ABB RobotStudio station: ProiectSCR.rspag

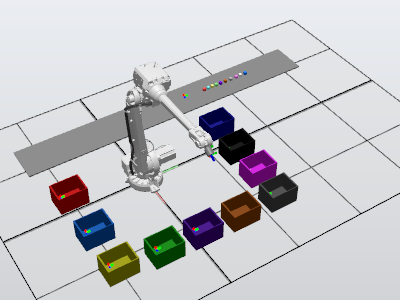
--- station ---
Station Tema1_SCR_Grigore_Vlad (saved by RobotStudio 24.3.10958.1)
Controller IRB4600_20_250
  mechanical unit ROB_1: IRB4600_20_250_C_01, 6 joints, base frame (0, 0, 0) mm
Layout (positions relative to the parent item):
  - IRB4600_20_250_C_01 [mechanism, from %ABB.RobotStudio.Models.IRB4600%\IRB4600_20_250_C_G_01.rslib] at (0, 0, 0) mm; joint values [0, 0, 0, 0, 0.5236, 0] (rad or m)
  - Container_1 [part] at (-320.44, -1190.22, 30) mm, size 300 x 400 x 270 mm
  - Banda [part] at (-1428.04, -1283.76, 0) mm, size 550 x 4550 x 20 mm
  - Pachet_1 [part] at (-1164.97, 1677.25, 60) mm, rotated rx 180 ry 0 rz 180 deg, size 40 x 40 x 40 mm
  - Container_2 [part] at (386.4, -1190.22, 30) mm, size 300 x 400 x 270 mm
  - Container_3 [part] at (1012.12, -1190.22, 30) mm, size 300 x 400 x 270 mm
  - Container_4 [part] at (1087.87, -610.7, 30) mm, size 300 x 400 x 270 mm
  - Container_6 [part] at (1101.15, 485.48, 30) mm, size 300 x 400 x 270 mm
  - Container_7 [part] at (1088.83, 1073.15, 30) mm, size 300 x 400 x 270 mm
  - Container_8 [part] at (596.46, 1111.34, 30) mm, size 300 x 400 x 270 mm
  - Container_9 [part] at (89.93, 1120.66, 30) mm, size 300 x 400 x 270 mm
  - Container_10 [part] at (-439.15, 1146.37, 30) mm, size 300 x 400 x 270 mm
  - MyNewTool [mechanism] at (1479.11, 0, 1722.5) mm, rotated rx 180 ry 60 rz 180 deg
      TCP MyNewTool at (0, 0, 80) mm
      links: Part_2
  - Container_5 [part] at (1087.87, -64.6, 30) mm, size 300 x 400 x 270 mm
  - Pachet_3 [part] at (-1164.97, 1820.33, 60) mm, rotated rx 180 ry 0 rz 180 deg, size 40 x 40 x 40 mm
  - Pachet_5 [part] at (-1164.97, 1973.31, 60) mm, rotated rx 180 ry 0 rz 180 deg, size 40 x 40 x 40 mm
  - Pachet_6 [part] at (-1164.97, 2058.75, 60) mm, rotated rx 180 ry 0 rz 180 deg, size 40 x 40 x 40 mm
  - Pachet_7 [part] at (-1164.97, 2158.23, 60) mm, rotated rx 180 ry 0 rz 180 deg, size 40 x 40 x 40 mm
  - Pachet_8 [part] at (-1164.97, 2259.91, 60) mm, rotated rx 180 ry 0 rz 180 deg, size 40 x 40 x 40 mm
  - Pachet_10 [part] at (-1164.97, 2429.71, 60) mm, rotated rx 180 ry 0 rz 180 deg, size 40 x 40 x 40 mm
  - Pachet_4 [part] at (-1164.97, 1892.62, 60) mm, rotated rx 180 ry 0 rz 180 deg, size 40 x 40 x 40 mm
  - Pachet_9 [part] at (-1164.97, 2336.17, 60) mm, rotated rx 180 ry 0 rz 180 deg, size 40 x 40 x 40 mm
  - SmartComponent_1 [smart component]
      signals: DI Get, DI DeleteAll
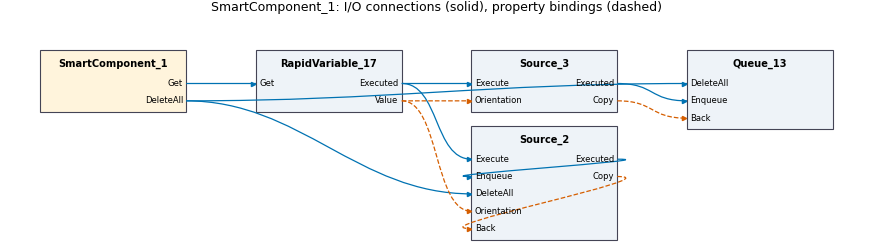
      connections:
        SmartComponent_1.Get -> RapidVariable_17.Get
        RapidVariable_17.Executed -> Source_2.Execute
        Source_2.Executed -> Queue_12.Enqueue
        SmartComponent_1.DeleteAll -> Queue_12.DeleteAll
        SmartComponent_1.DeleteAll -> Queue_13.DeleteAll
        Source_3.Executed -> Queue_13.Enqueue
        RapidVariable_17.Executed -> Source_3.Execute
        RapidVariable_17.Value => Source_2.Orientation
        Source_2.Copy => Queue_12.Back
        RapidVariable_17.Value => Source_3.Orientation
        Source_3.Copy => Queue_13.Back
    - RapidVariable_17 [smart component, from Components\RapidVariable.rslib]
        properties: DataType=orient; Controller=IRB4600_20_250; Task=T_ROB1; Module=Module1; Variable=RotXYZ; Value=[3.14159265358979 1.08734199990513E-38 3.14159265358979]
    - Source_3 [smart component, from Components\Source.rslib]
        properties: Source=Pachet_1; Copy=(none); Parent=(none); Position=[-1.164969 1.332694 0.06]; Orientation=[3.14159265358979 1.08734199990513E-38 3.14159265358979]; Transient=false; PhysicsBehavior=-1
    - Queue_13 [smart component, from Components\Queue.rslib]
        properties: Back=(none); Front=(none); Queue=; NumberOfObjects=0
  - SmartComponent_2 [smart component]
      signals: DI Get, DI DeleteAll
      connections:
        SmartComponent_2.Get -> RapidVariable_17.Get
        RapidVariable_17.Executed -> Source_2.Execute
        Source_2.Executed -> Queue_12.Enqueue
        SmartComponent_2.DeleteAll -> Queue_12.DeleteAll
        RapidVariable_17.Executed -> Source_4.Execute
        Source_4.Executed -> Queue_12.Enqueue
        RapidVariable_17.Value => Source_2.Orientation
        Source_2.Copy => Queue_12.Back
        RapidVariable_17.Value => Source_4.Orientation
        Source_4.Copy => Queue_12.Back
    - RapidVariable_17 [smart component, from Components\RapidVariable.rslib]
        properties: DataType=orient; Controller=IRB4600_20_250; Task=T_ROB1; Module=Module1; Variable=RotXYZ; Value=[3.14159265358979 1.08734199990513E-38 3.14159265358979]
    - Queue_12 [smart component, from Components\Queue.rslib]
        properties: Back=(none); Front=(none); Queue=; NumberOfObjects=0
    - Source_4 [smart component, from Components\Source.rslib]
        properties: Source=Pachet_2; Copy=(none); Parent=(none); Position=[-1.164969 1.332694 0.06]; Orientation=[3.14159265358979 1.08734199990513E-38 3.14159265358979]; Transient=false; PhysicsBehavior=-1
  - SmartComponent_3 [smart component]
      signals: DI Get, DI DeleteAll
      connections:
        SmartComponent_3.Get -> RapidVariable_17.Get
        RapidVariable_17.Executed -> Source_2.Execute
        Source_2.Executed -> Queue_12.Enqueue
        SmartComponent_3.DeleteAll -> Queue_12.DeleteAll
        RapidVariable_17.Value => Source_2.Orientation
        Source_2.Copy => Queue_12.Back
    - Source_2 [smart component, from Components\Source.rslib]
        properties: Source=Pachet_3; Copy=(none); Parent=(none); Position=[-1.164969 1.332694 0.06]; Orientation=[3.14159265358979 1.08734199990513E-38 3.14159265358979]; Transient=false; PhysicsBehavior=-1
    - RapidVariable_17 [smart component, from Components\RapidVariable.rslib]
        properties: DataType=orient; Controller=IRB4600_20_250; Task=T_ROB1; Module=Module1; Variable=RotXYZ; Value=[3.14159265358979 1.08734199990513E-38 3.14159265358979]
    - Queue_12 [smart component, from Components\Queue.rslib]
        properties: Back=(none); Front=(none); Queue=; NumberOfObjects=0
  - SmartComponent_4 [smart component]
      signals: DI Get, DI DeleteAll
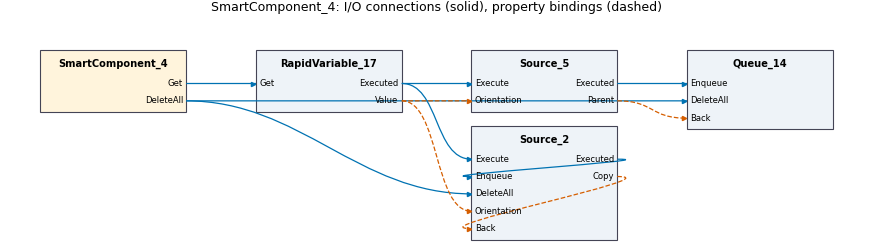
      connections:
        SmartComponent_4.Get -> RapidVariable_17.Get
        RapidVariable_17.Executed -> Source_2.Execute
        Source_2.Executed -> Queue_12.Enqueue
        SmartComponent_4.DeleteAll -> Queue_12.DeleteAll
        RapidVariable_17.Executed -> Source_5.Execute
        Source_5.Executed -> Queue_14.Enqueue
        SmartComponent_4.DeleteAll -> Queue_14.DeleteAll
        RapidVariable_17.Value => Source_2.Orientation
        Source_2.Copy => Queue_12.Back
        RapidVariable_17.Value => Source_5.Orientation
        Source_5.Parent => Queue_14.Back
    - RapidVariable_17 [smart component, from Components\RapidVariable.rslib]
        properties: DataType=orient; Controller=IRB4600_20_250; Task=T_ROB1; Module=Module1; Variable=RotXYZ; Value=[0 0 0]
    - Source_5 [smart component, from Components\Source.rslib]
        properties: Source=Pachet_4; Copy=(none); Parent=(none); Position=[-1.164969 1.332694 0.06]; Orientation=[0 0 0]; Transient=false; PhysicsBehavior=-1
    - Queue_14 [smart component, from Components\Queue.rslib]
        properties: Back=(none); Front=(none); Queue=; NumberOfObjects=0
  - SmartComponent_5 [smart component]
      signals: DI Get, DI DeleteAll
      connections:
        SmartComponent_5.Get -> RapidVariable_17.Get
        RapidVariable_17.Executed -> Source_2.Execute
        Source_2.Executed -> Queue_12.Enqueue
        SmartComponent_5.DeleteAll -> Queue_12.DeleteAll
        RapidVariable_17.Executed -> Source_6.Execute
        Source_6.Executed -> Queue_15.Enqueue
        SmartComponent_5.DeleteAll -> Queue_15.DeleteAll
        RapidVariable_17.Value => Source_2.Orientation
        Source_2.Copy => Queue_12.Back
        Source_6.Copy => Queue_15.Back
        RapidVariable_17.Value => Source_6.Orientation
    - RapidVariable_17 [smart component, from Components\RapidVariable.rslib]
        properties: DataType=orient; Controller=IRB4600_20_250; Task=T_ROB1; Module=Module1; Variable=RotXYZ; Value=[0 0 0]
    - Source_6 [smart component, from Components\Source.rslib]
        properties: Source=Pachet_5; Copy=(none); Parent=(none); Position=[-1.164969 1.332694 0.06]; Orientation=[0 0 0]; Transient=false; PhysicsBehavior=-1
    - Queue_15 [smart component, from Components\Queue.rslib]
        properties: Back=(none); Front=(none); Queue=; NumberOfObjects=0
  - SmartComponent_6 [smart component]
      signals: DI Get, DI DeleteAll
      connections:
        SmartComponent_6.Get -> RapidVariable_17.Get
        RapidVariable_17.Executed -> Source_2.Execute
        Source_2.Executed -> Queue_12.Enqueue
        SmartComponent_6.DeleteAll -> Queue_12.DeleteAll
        RapidVariable_17.Executed -> Source_7.Execute
        Source_7.Executed -> Queue_16.Enqueue
        SmartComponent_6.DeleteAll -> Queue_16.DeleteAll
        RapidVariable_17.Value => Source_2.Orientation
        Source_2.Copy => Queue_12.Back
        Source_7.Copy => Queue_16.Back
        RapidVariable_17.Value => Source_7.Orientation
    - RapidVariable_17 [smart component, from Components\RapidVariable.rslib]
        properties: DataType=orient; Controller=IRB4600_20_250; Task=T_ROB1; Module=Module1; Variable=RotXYZ; Value=[0 0 0]
    - Source_7 [smart component, from Components\Source.rslib]
        properties: Source=Pachet_6; Copy=(none); Parent=(none); Position=[-1.164969 1.332694 0.06]; Orientation=[0 0 0]; Transient=false; PhysicsBehavior=-1
    - Queue_16 [smart component, from Components\Queue.rslib]
        properties: Back=(none); Front=(none); Queue=; NumberOfObjects=0
  - SmartComponent_7 [smart component]
      signals: DI Get, DI DeleteAll
      connections:
        SmartComponent_7.Get -> RapidVariable_17.Get
        RapidVariable_17.Executed -> Source_2.Execute
        Source_2.Executed -> Queue_12.Enqueue
        SmartComponent_7.DeleteAll -> Queue_12.DeleteAll
        RapidVariable_17.Executed -> Source_8.Execute
        Source_8.Executed -> Queue_17.Enqueue
        SmartComponent_7.DeleteAll -> Queue_17.DeleteAll
        RapidVariable_17.Value => Source_2.Orientation
        Source_2.Copy => Queue_12.Back
        Source_8.Copy => Queue_17.Back
        RapidVariable_17.Value => Source_8.Orientation
    - RapidVariable_17 [smart component, from Components\RapidVariable.rslib]
        properties: DataType=orient; Controller=IRB4600_20_250; Task=T_ROB1; Module=Module1; Variable=RotXYZ; Value=[0 0 0]
    - Source_8 [smart component, from Components\Source.rslib]
        properties: Source=Pachet_7; Copy=(none); Parent=(none); Position=[-1.164969 1.332694 0.06]; Orientation=[0 0 0]; Transient=false; PhysicsBehavior=-1
    - Queue_17 [smart component, from Components\Queue.rslib]
        properties: Back=(none); Front=(none); Queue=; NumberOfObjects=0
  - SmartComponent_8 [smart component]
      signals: DI Get, DI DeleteAll
      connections:
        SmartComponent_8.Get -> RapidVariable_17.Get
        RapidVariable_17.Executed -> Source_2.Execute
        Source_2.Executed -> Queue_12.Enqueue
        SmartComponent_8.DeleteAll -> Queue_12.DeleteAll
        RapidVariable_17.Executed -> Source_10.Execute
        Source_10.Executed -> Queue_18.Enqueue
        SmartComponent_8.DeleteAll -> Queue_18.DeleteAll
        RapidVariable_17.Value => Source_2.Orientation
        Source_2.Copy => Queue_12.Back
        RapidVariable_17.Value => Source_10.Orientation
        Source_10.Copy => Queue_18.Back
    - RapidVariable_17 [smart component, from Components\RapidVariable.rslib]
        properties: DataType=orient; Controller=IRB4600_20_250; Task=T_ROB1; Module=Module1; Variable=RotXYZ; Value=[0 0 0]
    - Source_10 [smart component, from Components\Source.rslib]
        properties: Source=Pachet_8; Copy=(none); Parent=(none); Position=[-1.164969 1.332694 0.06]; Orientation=[0 0 0]; Transient=false; PhysicsBehavior=-1
    - Queue_18 [smart component, from Components\Queue.rslib]
        properties: Back=(none); Front=(none); Queue=; NumberOfObjects=0
  - SmartComponent_9 [smart component]
      signals: DI Get, DI DeleteAll
      connections:
        SmartComponent_9.Get -> RapidVariable_17.Get
        RapidVariable_17.Executed -> Source_2.Execute
        Source_2.Executed -> Queue_12.Enqueue
        SmartComponent_9.DeleteAll -> Queue_12.DeleteAll
        RapidVariable_17.Executed -> Source_11.Execute
        Source_11.Executed -> Queue_19.Enqueue
        SmartComponent_9.DeleteAll -> Queue_19.DeleteAll
        RapidVariable_17.Value => Source_2.Orientation
        Source_2.Copy => Queue_12.Back
        Source_11.Copy => Queue_19.Back
        RapidVariable_17.Value => Source_11.Orientation
    - RapidVariable_17 [smart component, from Components\RapidVariable.rslib]
        properties: DataType=orient; Controller=IRB4600_20_250; Task=T_ROB1; Module=Module1; Variable=RotXYZ; Value=[0 0 0]
    - Source_11 [smart component, from Components\Source.rslib]
        properties: Source=Pachet_9; Copy=(none); Parent=(none); Position=[-1.164969 1.332694 0.06]; Orientation=[0 0 0]; Transient=false; PhysicsBehavior=-1
    - Queue_19 [smart component, from Components\Queue.rslib]
        properties: Back=(none); Front=(none); Queue=; NumberOfObjects=0
  - SmartComponent_10 [smart component]
      signals: DI Get, DI DeleteAll
      connections:
        SmartComponent_10.Get -> RapidVariable_17.Get
        RapidVariable_17.Executed -> Source_2.Execute
        Source_2.Executed -> Queue_12.Enqueue
        SmartComponent_10.DeleteAll -> Queue_12.DeleteAll
        RapidVariable_17.Executed -> Source_13.Execute
        Source_13.Executed -> Queue_20.Enqueue
        SmartComponent_10.DeleteAll -> Queue_20.DeleteAll
        RapidVariable_17.Value => Source_2.Orientation
        Source_2.Copy => Queue_12.Back
        Source_13.Copy => Queue_20.Back
        RapidVariable_17.Value => Source_13.Orientation
    - RapidVariable_17 [smart component, from Components\RapidVariable.rslib]
        properties: DataType=orient; Controller=IRB4600_20_250; Task=T_ROB1; Module=Module1; Variable=RotXYZ; Value=[0 0 0]
    - Source_13 [smart component, from Components\Source.rslib]
        properties: Source=Pachet_10; Copy=(none); Parent=(none); Position=[-1.164969 1.332694 0.06]; Orientation=[0 0 0]; Transient=false; PhysicsBehavior=-1
    - Queue_20 [smart component, from Components\Queue.rslib]
        properties: Back=(none); Front=(none); Queue=; NumberOfObjects=0
  - Pachet_2 [part] at (-1164.97, 1747.44, 60) mm, rotated rx 180 ry 0 rz 180 deg, size 40 x 40 x 40 mm
Attachment: MyNewTool is attached to IRB4600_20_250_C_01 / Link6
EventTableEntry 2341: ActivationMode=2, Cyclic=false, Group=, Trigger=aa_gripper 2342, Actions=[EventTableActionAttach 2343], Comment=
EventTableTriggerIO 2342: Operator=0, IOValue=[1], IRC5Controller=? -1, SignalSource=IRB4600_20_250 1196
EventTableActionAttach 2343: MountObject=true, FlangeIndext=0, FindNearest=true, AttachmentParent=MyNewTool 2337, AttachmentChild=? -1, Offset=[X=1, Y=0, Z=0, W=0, X=0, Y=1, Z=0, W=0, X=0, Y=0, Z=1, W=0, X=0, Y=0, Z=0, W=1]
EventTableEntry 2344: ActivationMode=2, Cyclic=false, Group=, Trigger=aa_gripper 2345, Actions=[EventTableActionDetach 2346], Comment=
EventTableTriggerIO 2345: Operator=0, IOValue=[0], IRC5Controller=? -1, SignalSource=IRB4600_20_250 1196
EventTableActionDetach 2346: AttachmentParent=MyNewTool 2337, AttachmentChild=? -1
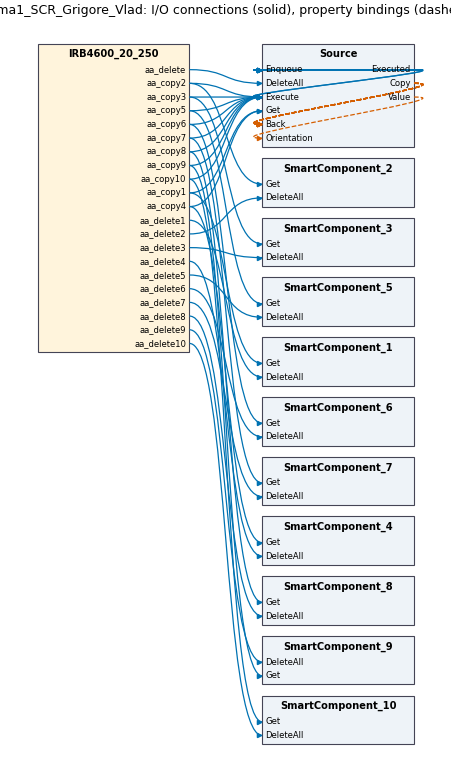
Station logic (signal -> signal, property => property):
  Source.Executed -> Queue.Enqueue
  IRB4600_20_250.aa_delete -> Queue.DeleteAll
  IRB4600_20_250.aa_copy2 -> Source_2.Execute
  Source_2.Executed -> Queue.Enqueue
  IRB4600_20_250.aa_copy3 -> Source_3.Execute
  Source_3.Executed -> Queue.Enqueue
  Source_4.Executed -> Queue.Enqueue
  IRB4600_20_250.aa_copy5 -> Source_5.Execute
  Source_5.Executed -> Queue.Enqueue
  IRB4600_20_250.aa_copy6 -> Source_6.Execute
  Source_6.Executed -> Queue.Enqueue
  IRB4600_20_250.aa_copy7 -> Source_7.Execute
  Source_7.Executed -> Queue.Enqueue
  IRB4600_20_250.aa_copy8 -> Source_8.Execute
  Source_8.Executed -> Queue.Enqueue
  IRB4600_20_250.aa_copy9 -> Source_9.Execute
  Source_9.Executed -> Queue.Enqueue
  IRB4600_20_250.aa_copy10 -> Source_10.Execute
  Source_10.Executed -> Queue.Enqueue
  IRB4600_20_250.aa_copy1 -> RapidVariable.Get
  RapidVariable.Executed -> Source.Execute
  Source.Executed -> Queue.Enqueue
  IRB4600_20_250.aa_copy4 -> RapidVariable_4.Get
  RapidVariable_4.Executed -> Source_4.Execute
  Source_4.Executed -> Queue_4.Enqueue
  IRB4600_20_250.aa_copy1 -> SmartComponent_1.Get
  IRB4600_20_250.aa_delete1 -> SmartComponent_1.DeleteAll
  IRB4600_20_250.aa_copy2 -> SmartComponent_2.Get
  IRB4600_20_250.aa_delete2 -> SmartComponent_2.DeleteAll
  IRB4600_20_250.aa_copy3 -> SmartComponent_3.Get
  IRB4600_20_250.aa_delete3 -> SmartComponent_3.DeleteAll
  IRB4600_20_250.aa_copy4 -> SmartComponent_4.Get
  IRB4600_20_250.aa_delete4 -> SmartComponent_4.DeleteAll
  IRB4600_20_250.aa_copy5 -> SmartComponent_5.Get
  IRB4600_20_250.aa_delete5 -> SmartComponent_5.DeleteAll
  IRB4600_20_250.aa_copy6 -> SmartComponent_6.Get
  IRB4600_20_250.aa_delete6 -> SmartComponent_6.DeleteAll
  IRB4600_20_250.aa_copy7 -> SmartComponent_7.Get
  IRB4600_20_250.aa_delete7 -> SmartComponent_7.DeleteAll
  IRB4600_20_250.aa_copy8 -> SmartComponent_8.Get
  IRB4600_20_250.aa_delete8 -> SmartComponent_8.DeleteAll
  IRB4600_20_250.aa_delete9 -> SmartComponent_9.DeleteAll
  IRB4600_20_250.aa_copy9 -> SmartComponent_9.Get
  IRB4600_20_250.aa_copy10 -> SmartComponent_10.Get
  IRB4600_20_250.aa_delete10 -> SmartComponent_10.DeleteAll
  Source.Copy => Queue.Back
  Source_2.Copy => Queue.Back
  Source_3.Copy => Queue.Back
  Source_4.Copy => Queue.Back
  Source_5.Copy => Queue.Back
  Source_6.Copy => Queue.Back
  Source_8.Copy => Queue.Back
  Source_9.Copy => Queue.Back
  Source_10.Copy => Queue.Back
  Source.Copy => Queue.Back
  RapidVariable.Value => Source.Orientation
  Source_4.Copy => Queue_4.Back

--- Controller Data/IRB4600_20_250/RAPID/TASK1/PROGMOD/CalibData.mod ---
MODULE CalibData
    PERS tooldata MyNewTool:=[TRUE,[[0,0,80],[1,0,0,0]],[1,[0,0,1],[1,0,0,0],0,0,0]];
    TASK PERS wobjdata Container_1:=[FALSE,TRUE,"",[[-320.441,-1190.22,30],[1,0,0,0]],[[0,0,0],[1,0,0,0]]];
ENDMODULE

--- Controller Data/IRB4600_20_250/RAPID/TASK1/PROGMOD/Module1.mod ---
MODULE Module1
        CONST robtarget Home:=[[1548.394191624,0,1682.5],[0.5,0,0.866025404,0],[0,0,0,0],[9E+09,9E+09,9E+09,9E+09,9E+09,9E+09]];
    VAR robtarget Pick:=[[-1164.969,1332.694,60],[0,0,1,0],[1,0,1,0],[9E+09,9E+09,9E+09,9E+09,9E+09,9E+09]];
    VAR robtarget Place_1:=[[-244.846202712,-1105.356578591,70],[0,0,1,0],[-2,0,-2,0],[9E+09,9E+09,9E+09,9E+09,9E+09,9E+09]];
    VAR robtarget my_place;
    VAR robtarget my_pick;
    VAR robtarget Place_2:=[[460.463358068,-1090.594225612,70],[0,0,1,0],[-1,0,-1,0],[9E+09,9E+09,9E+09,9E+09,9E+09,9E+09]];
    VAR robtarget Place_3:=[[1075.470180633,-1093.870090064,70],[0,0,1,0],[-1,0,-1,0],[9E+09,9E+09,9E+09,9E+09,9E+09,9E+09]];
    VAR robtarget Place_4:=[[1155.434000146,-497.782325439,70],[0,0,1,0],[-1,0,-1,0],[9E+09,9E+09,9E+09,9E+09,9E+09,9E+09]];
    VAR robtarget Place_5:=[[1148.232307595,45.80205686,70],[0,0,1,0],[0,0,0,0],[9E+09,9E+09,9E+09,9E+09,9E+09,9E+09]];
    VAR robtarget Place_6:=[[1155.662806581,542.759763513,70],[0,0,1,0],[0,0,0,0],[9E+09,9E+09,9E+09,9E+09,9E+09,9E+09]];
    VAR robtarget Place_7:=[[1142.490790536,1166.144270434,70],[0,0,1,0],[0,0,0,0],[9E+09,9E+09,9E+09,9E+09,9E+09,9E+09]];
    VAR robtarget Place_8:=[[652.5146322,1189.626758644,70],[0,0,1,0],[0,0,0,0],[9E+09,9E+09,9E+09,9E+09,9E+09,9E+09]];
    VAR robtarget Place_9:=[[148.244670469,1200.420807904,70],[0,0,1,0],[0,0,0,0],[9E+09,9E+09,9E+09,9E+09,9E+09,9E+09]];
    VAR robtarget Place_10:=[[-377.052456308,1219.115498151,70],[0,0,1,0],[1,0,1,0],[9E+09,9E+09,9E+09,9E+09,9E+09,9E+09]];
    VAR socketdev client;
    VAR string tip_piesa;
    VAR string rot_x;
    VAR string rot_y;
    VAR string rot_z;
    VAR num x_rot;
    VAR num y_rot;
    VAR num z_rot;
    VAR bool succes;
    VAR num i1;
    VAR num i2;
    VAR num i3;
    VAR num i4;
    VAR num i5;
    VAR num i6;
    VAR num i7;
    VAR num i8;
    VAR num i9;
    VAR num i10;
    VAR orient RotXYZ;
!***********************************************************
    !
    ! Module:  Module1
    !
    ! Description:
    !   <Insert description here>
    !
    ! Author: Asus
    !
    ! Version: 1.0
    !
    !***********************************************************


    !***********************************************************
    !
    ! Procedure main
    !
    !   This is the entry point of your program
    !
    !***********************************************************
    PROC main()
        !Add your code here
        ! Bucla infinita deoarece vrem sa putem pune si alte optiuni fara sa se termine de rulat programul
        i1 := 0;
        i2 := 0;
        i3 := 0;
        i4 := 0;
        i5 := 0;
        i6 := 0;
        i7 := 0;
        i8 := 0;
        i9 := 0;
        i10 := 0;
        WHILE TRUE DO
            msj_client;
            IF tip_piesa = "Piesa_1" THEN
                ! Spatiu
                SetDO aa_gripper, 0;
                SetDO aa_copy1,0;
                SetDO aa_delete1, 0;
                MoveJ Home,v1000,fine,MyNewTool\WObj:=wobj0;

                rotatie;
                RotXYZ := OrientZYX(180 - z_rot, - y_rot, 180 - x_rot );
                Pick.rot := RotXYZ;
                my_pick := Pick;
                SetDO aa_copy1,1;

                my_place := offs(Place_1, ( i1 MOD 4) * 50, (( i1 DIV 4 ) MOD 3 ) * 50, -( i1 DIV 12 ) * 50 );
                pick_and_place;
                i1 := i1 + 1;
                SetDO aa_copy1,0;

                MoveJ Home,v1000,fine,MyNewTool\WObj:=wobj0;

                IF i1 = 23 THEN
                    SetDO aa_delete1, 1;
                    i1 := 0;
                ENDIF

            ELSEIF tip_piesa = "Piesa_2" THEN
                !Spatiu
                SetDO aa_gripper, 0;
                SetDO aa_copy2,0;
                SetDO aa_delete2, 0;
                MoveJ Home,v1000,fine,MyNewTool\WObj:=wobj0;

                rotatie;
                RotXYZ := OrientZYX(180 - z_rot, - y_rot, 180 - x_rot );
                Pick.rot := RotXYZ;
                my_pick := Pick;
                SetDO aa_copy2,1;

                my_place := offs(Place_2, ( i2 MOD 4) * 50, (( i2 DIV 4 ) MOD 3 ) * 50, -( i2 DIV 12 ) * 50 );
                pick_and_place;
                i2 := i2 + 1;
                SetDO aa_copy2,0;

                MoveJ Home,v1000,fine,MyNewTool\WObj:=wobj0;

                IF i2 = 23 THEN
                    SetDO aa_delete2, 1;
                    i2 := 0;
                ENDIF

            ELSEIF tip_piesa = "Piesa_3" THEN
                !Spatiu
                SetDO aa_gripper, 0;
                SetDO aa_copy3,0;
                SetDO aa_delete3, 0;
                MoveJ Home,v1000,fine,MyNewTool\WObj:=wobj0;

                rotatie;
                RotXYZ := OrientZYX(180 - z_rot, - y_rot, 180 - x_rot );
                Pick.rot := RotXYZ;
                my_pick := Pick;
                SetDO aa_copy3,1;

                my_place := offs(Place_3, ( i3 MOD 4) * 50, (( i3 DIV 4 ) MOD 3 ) * 50, -( i3 DIV 12 ) * 50 );
                pick_and_place;
                i3 := i3 + 1;
                SetDO aa_copy3,0;

                MoveJ Home,v1000,fine,MyNewTool\WObj:=wobj0;

                IF i3 = 23 THEN
                    SetDO aa_delete3, 1;
                    i3 := 0;
                ENDIF

             ELSEIF tip_piesa = "Piesa_4" THEN
                !Spatiu
                SetDO aa_gripper, 0;
                SetDO aa_copy4,0;
                SetDO aa_delete4, 0;
                MoveJ Home,v1000,fine,MyNewTool\WObj:=wobj0;

                rotatie;
                RotXYZ := OrientZYX(180 - z_rot, - y_rot, 180 - x_rot );
                Pick.rot := RotXYZ;
                my_pick := Pick;
                SetDO aa_copy4,1;

                my_place := Offs(Place_4, ( i4 MOD 4) * 50, (( i4 DIV 4 ) MOD 3 ) * 50, -( i4 DIV 12 ) * 50 );
                pick_and_place;
                i4 := i4 + 1;
                SetDO aa_copy4,0;

                MoveJ Home,v1000,fine,MyNewTool\WObj:=wobj0;

                IF i4 = 23 THEN
                    SetDO aa_delete4, 1;
                    i4 := 0;
                ENDIF

             ELSEIF tip_piesa = "Piesa_5" THEN
                !Spatiu
                SetDO aa_gripper, 0;
                SetDO aa_copy5,0;
                SetDO aa_delete5, 0;
                MoveJ Home,v1000,fine,MyNewTool\WObj:=wobj0;

                rotatie;
                RotXYZ := OrientZYX(180 - z_rot, - y_rot, 180 - x_rot );
                Pick.rot := RotXYZ;
                my_pick := Pick;
                SetDO aa_copy5,1;

                my_place := offs(Place_5, ( i5 MOD 4) * 50, (( i5 DIV 4 ) MOD 3 ) * 50, -( i5 DIV 12 ) * 50 );
                pick_and_place;
                i5 := i5 + 1;
                SetDO aa_copy5,0;

                MoveJ Home,v1000,fine,MyNewTool\WObj:=wobj0;

                IF i5 = 23 THEN
                    SetDO aa_delete5, 1;
                    i5 := 0;
                ENDIF

            ELSEIF tip_piesa = "Piesa_6" THEN
                !Spatiu
                SetDO aa_gripper, 0;
                SetDO aa_copy6,0;
                SetDO aa_delete6, 0;
                MoveJ Home,v1000,fine,MyNewTool\WObj:=wobj0;

                rotatie;
                RotXYZ := OrientZYX(180 - z_rot, - y_rot, 180 - x_rot );
                Pick.rot := RotXYZ;
                my_pick := Pick;
                SetDO aa_copy6,1;

                my_place := offs(Place_6, ( i6 MOD 4) * 50, (( i6 DIV 4 ) MOD 3 ) * 50, -( i6 DIV 12 ) * 50 );
                pick_and_place;
                i6 := i6 + 1;
                SetDO aa_copy6,0;

                MoveJ Home,v1000,fine,MyNewTool\WObj:=wobj0;

                IF i6 = 23 THEN
                    SetDO aa_delete6, 1;
                    i6 := 0;
                ENDIF

            ELSEIF tip_piesa = "Piesa_7" THEN
                !Spatiu
                SetDO aa_gripper, 0;
                SetDO aa_copy7,0;
                SetDO aa_delete7, 0;
                MoveJ Home,v1000,fine,MyNewTool\WObj:=wobj0;

                rotatie;
                RotXYZ := OrientZYX(180 - z_rot, - y_rot, 180 - x_rot );
                Pick.rot := RotXYZ;
                my_pick := Pick;
                SetDO aa_copy7,1;

                my_place := offs(Place_7, ( i7 MOD 4) * 50, (( i7 DIV 4 ) MOD 3 ) * 50, -( i7 DIV 12 ) * 50 );
                pick_and_place;
                i7 := i7 + 1;
                SetDO aa_copy7,0;

                MoveJ Home,v1000,fine,MyNewTool\WObj:=wobj0;

                IF i7 = 23 THEN
                    SetDO aa_delete7, 1;
                    i7 := 0;
                ENDIF

            ELSEIF tip_piesa = "Piesa_8" THEN
                !Spatiu
                SetDO aa_gripper, 0;
                SetDO aa_copy8,0;
                SetDO aa_delete8, 0;
                MoveJ Home,v1000,fine,MyNewTool\WObj:=wobj0;

                rotatie;
                RotXYZ := OrientZYX(180 - z_rot, - y_rot, 180 - x_rot );
                Pick.rot := RotXYZ;
                my_pick := Pick;
                SetDO aa_copy8,1;

                my_place := offs(Place_8, ( i8 MOD 4) * 50, (( i8 DIV 4 ) MOD 3 ) * 50, -( i8 DIV 12 ) * 50 );
                pick_and_place;
                i8 := i8 + 1;
                SetDO aa_copy8, 0;

                MoveJ Home,v1000,fine,MyNewTool\WObj:=wobj0;

                IF i8 = 23 THEN
                    SetDO aa_delete8, 1;
                    i8 := 0;
                ENDIF

            ELSEIF tip_piesa = "Piesa_9" THEN
                !Spatiu
                SetDO aa_gripper, 0;
                SetDO aa_copy9,0;
                SetDO aa_delete9, 0;
                MoveJ Home,v1000,fine,MyNewTool\WObj:=wobj0;

                rotatie;
                RotXYZ := OrientZYX(180 - z_rot, - y_rot, 180 - x_rot );
                Pick.rot := RotXYZ;
                my_pick := Pick;
                SetDO aa_copy9,1;

                my_place := offs(Place_9, ( i9 MOD 4) * 50, (( i9 DIV 4 ) MOD 3 ) * 50, -( i9 DIV 12 ) * 50 );
                pick_and_place;
                i9 := i9 + 1;
                SetDO aa_copy9, 0;

                MoveJ Home,v1000,fine,MyNewTool\WObj:=wobj0;

                IF i9 = 23 THEN
                    SetDO aa_delete9, 1;
                    i9 := 0;
                ENDIF

            ELSEIF tip_piesa = "Piesa_10" THEN
                !Spatiu
                SetDO aa_gripper, 0;
                SetDO aa_copy10,0;
                SetDO aa_delete10, 0;
                MoveJ Home,v1000,fine,MyNewTool\WObj:=wobj0;

                rotatie;
                RotXYZ := OrientZYX(180 - z_rot, - y_rot, 180 - x_rot );
                Pick.rot := RotXYZ;
                my_pick := Pick;
                SetDO aa_copy10,1;

                my_place := offs(Place_10, ( i10 MOD 4) * 50, (( i10 DIV 4 ) MOD 3 ) * 50, -( i10 DIV 12 ) * 50 );
                pick_and_place;
                i10 := i10 + 1;
                SetDO aa_copy10, 0;

                MoveJ Home,v1000,fine,MyNewTool\WObj:=wobj0;

                 IF i10 = 23 THEN
                    i10 := 0;
                ENDIF

            ENDIF
        ENDWHILE
        SetDO aa_delete10,1;
    ENDPROC
    PROC pick_and_place()
        MoveJ offs(my_pick, 0, 0, 100),v1000,fine,MyNewTool\WObj:=wobj0;
        MoveL my_pick,v1000,fine,MyNewTool\WObj:=wobj0;
        SetDO aa_gripper, 1;
        WaitTime 0.5;
        MoveL offs(my_pick, 0, 0, 100),v1000,fine,MyNewTool\WObj:=wobj0;

        MoveJ offs(my_place, 0, 0, 450),v1000,fine,MyNewTool\WObj:=wobj0;
        MoveL my_place,v1000,fine,MyNewTool\WObj:=wobj0;
        SetDO aa_gripper, 0;
        WaitTime 0.5;
        MoveL offs(my_place, 0, 0, 450),v1000,fine,MyNewTool\WObj:=wobj0;
    ENDPROC
    PROC msj_client()
        SocketSend client \Str:="Tip piesa:";
        SocketReceive client \Str:=tip_piesa;
        TPWrite "Selectie tip piesa";
        ERROR
        IF ERRNO = ERR_SOCK_TIMEOUT THEN
            RETRY;
        ELSEIF ERRNO = ERR_SOCK_CLOSED THEN
            ref_conexiune;
            RETRY;
        ELSE
            !err
        ENDIF
    ENDPROC
    PROC ref_conexiune()
        SocketClose client;
        SocketCreate client;
        SocketConnect client, "127.0.0.1", 1401;

         ERROR
        IF ERRNO = ERR_SOCK_TIMEOUT THEN
            RETRY;
        ELSEIF ERRNO = ERR_SOCK_CLOSED THEN
            RETURN;
        ELSE
            !err
        ENDIF
    ENDPROC
    PROC rotatie()
        SocketSend client \Str:="Rotatie Z:";
        SocketReceive client \Str:=rot_z;
        SocketSend client \Str:="Rotatie Y:";
        SocketReceive client \Str:=rot_y;
        SocketSend client \Str:="Rotatie X:";
        SocketReceive client \Str:=rot_x;
        succes := StrToVal(rot_z, z_rot);
        succes := StrToVal(rot_y, y_rot);
        succes := StrToVal(rot_x, x_rot);
        TPWrite "Rotatie";
        ERROR
        IF ERRNO = ERR_SOCK_TIMEOUT THEN
            RETRY;
        ELSEIF ERRNO = ERR_SOCK_CLOSED THEN
            ref_conexiune;
            RETRY;
        ELSE
            !err
        ENDIF
    ENDPROC
ENDMODULE

--- Controller Data/IRB4600_20_250/SYSPAR/EIO.cfg ---
EIO:CFG_1.0:6:1::
#
EIO_SIGNAL:

      -Name "aa_copy1" -SignalType "DO" -Access "All"

      -Name "aa_copy2" -SignalType "DO" -Access "All"

      -Name "aa_copy3" -SignalType "DO" -Access "All"

      -Name "aa_copy4" -SignalType "DO" -Access "All"

      -Name "aa_copy5" -SignalType "DO" -Access "All"

      -Name "aa_copy6" -SignalType "DO" -Access "All"

      -Name "aa_copy7" -SignalType "DO" -Access "All"

      -Name "aa_copy8" -SignalType "DO" -Access "All"

      -Name "aa_copy9" -SignalType "DO" -Access "All"

      -Name "aa_copy10" -SignalType "DO" -Access "All"

      -Name "aa_gripper" -SignalType "DO" -Access "All"

      -Name "aa_delete1" -SignalType "DO" -Access "All"

      -Name "aa_delete2" -SignalType "DO" -Access "All"

      -Name "aa_delete3" -SignalType "DO" -Access "All"

      -Name "aa_delete4" -SignalType "DO" -Access "All"

      -Name "aa_delete5" -SignalType "DO" -Access "All"

      -Name "aa_delete6" -SignalType "DO" -Access "All"

      -Name "aa_delete7" -SignalType "DO" -Access "All"

      -Name "aa_delete8" -SignalType "DO" -Access "All"

      -Name "aa_delete9" -SignalType "DO" -Access "All"

      -Name "aa_delete10" -SignalType "DO" -Access "All"
